{attribute 'qualified_only'}
VAR_GLOBAL
	// IM2L1-PPM-MMS
    {attribute 'pytmc' := 'pv: IM2L1:PPM:MMS'}
    {attribute 'TcLinkTo' := '.bLimitForwardEnable  := TIIB[IM2L1-EL7041]^STM Status^Status^Digital input 1;
                              .bLimitBackwardEnable := TIIB[IM2L1-EL7041]^STM Status^Status^Digital input 2;
                              .bBrakeRelease        := TIIB[IM2L1-EL2004]^Channel 1^Output'}
    M1: DUT_MotionStage := (sName := 'IM2L1:PPM:MMS');
END_VAR

(* stored: Version 1.1.0.1, ProductVersion 3.1.4024.6
   GVL Main: Id {f24be19c-614f-40ca-920f-63ab753550b2} *)
